Universal Robots PolyScope program: ReachV1Proj.urp

Program ReachV0Proj (installation=default directory=/home/ur/ursim-current/programs createdIn=5.8.0.10253 lastSavedIn=5.8.0.10253 robotSerialNumber=20195399999)
Calibrated DH parameters: a=[0, -0.24355, -0.2132, 0, 0, 0]; d=[0.15185, 0, 0, 0.13105, 0.08535, 0.0921]; alpha=[1.570796, 0, 0, 1.570796, -1.570796, 0]; deltaTheta=[0, 0, 0, 0, 0, 0]
Robot Program (runOnlyOnce=false)
  Script file /home/ur/ursim-current/programs/ReachV0.script
    | v = 0.25
    | a = 0.5
    | pose_init = [-1.57, -1.744, 1.57, -1.573, -1.573, -1.923]
    | global ready = False
    | write_output_integer_register(0, 0)
    | 
    | def inicio():
    |     global joints =  pose_init
    |     movej(joints, a, v)
    |     ready = True
    |     global flag = False
    |     write_output_integer_register(0, 1)
    | end
    | 
    | def updateActionRTDE():
    |     global action = [-1.57, -1.744, 1.57, -1.573, -1.573, -1.923]
    |     i=0
    |     while i<6:
    |         action[i] = read_input_float_register(i)
    |         i = i + 1
    |     end
    |     return action
    | end
    | 
    | # Definicion del programa principal.
    | def main_program():
    |     while ready == False or get_digital_out(2) == False or read_input_integer_register(0) == 0:
    |         if(ready == False):
    |             inicio()
    |         else:
    |             sync()
    |         end
    |     end
    |     while get_digital_out(2) == True and read_input_integer_register(0) == 1:
    |         sync()
    |         global flag = True
    |         joints = updateActionRTDE()
    |         servoj(joints, t=0.01, gain=20)
    |     end
    |     write_output_integer_register(0, 0)
    |     sync()
    | end
    | 
    | main_program()
